KUKA KRL program: cell.src

&ACCESS RVP
&REL 20
&COMMENT 03-10-R1 AUTO EXTERNAL MAIN
DEF  CELL ( )
;********************************
; Gestamp Standards
; Line - BMW G65 (cell 03)
; Robot 03-10-R1 (BMW-03-10-R1)
; Application - AUTOMATIC EXTERNAL MAIN PROGRAM (AUTOMATIONCORE CELL)
;********************************
;FOLD Initialize System
  ;NOTE: DMY IS A REMNANT OF THE KUKA CELL TEMPLATE (cellVorgabe): WRITTEN HERE, NEVER READ
  DECL CHAR DMY[3]
  DMY[]="---"
  ;AUTOMATIONCORE START-UP (HomeCheck, PROCESS RESET), THEN PTP TO HOME (HOME.src, P1 = XHOME)
  InitializeSystem()
  HOME()
  ;ENDFOLD (Initialize System)
  LOOP
    ;FOLD Maintain System
    ;RESET CYCLE DATA AND THE PLC HANDSHAKE OUTPUTS TO THEIR REST STATE (MaintainSystem), E.G.
    ;SIGNALS $OUT[5] do005RobotInCycle OFF, $OUT[15] do015WorkComplete OFF,
    ;$OUT[4] do004ProcessFault OFF, $OUT[141] do141RedRabbitFailed OFF,
    ;$OUT[142] do142RedRabbitPassed OFF; THEN WAITS HERE WHILE STOP AT END OF CYCLE IS
    ;SELECTED (SIGNAL $IN[147] di147SEOC ON, OR SELECTED BY THE USER)
    MaintainSystem()
    ;ENDFOLD (Maintain System)
    ;FOLD Check Style
    ;READ THE STYLE NUMBER - SIGNALS $IN[33..37] gdiStyle, ECHOED ON $OUT[33..37] gdoStyleAckn
    nStyle=gdiStyle
    gdoStyleAckn=nStyle
    ;READ THE OPTION NUMBER - SIGNALS $IN[38..45] gdiOption, ECHOED ON $OUT[38..45] gdoOptionAckn
    nOption=gdiOption
    gdoOptionAckn=nOption
    ;DECODE nOption INTO bOption1..8 (GetOptions) AND WRITE THEM TO
    ;SIGNALS $OUT[38..45] do038OptionAckn1..do045OptionAckn8
    GetOptions( )
    ;SHOW THE LAST CYCLE TIME AS A STATE MESSAGE
    GetCycTime( )
    ;FOLD State Message - Waiting for Cycle Start or Style Selection.
    IF (Exists_KrlMsg(nCycleStart_Handle)==FALSE) THEN
    	nCycleStart_Handle = Set_Krlmsg (#STATE, AutomationCore_Msg[24], AutoCore_MsgPar[], AutoCore_MsgOpt_NoStop)
    ENDIF
    ;ENDFOLD (State Message - Waiting for Cycle Start or Style Selection.)
    ;ENDFOLD (Check Style)
    ;CYCLE START - SIGNAL $IN[5] di005InitiateCycle ON, WITH nStyle > 0 AND nOption > 0
    IF ((di005InitiateCycle==TRUE) AND (nStyle>0) AND (nOption>0)) THEN
	    ;FOLD Start Cycle
	    ;CLEAR AUTOMATIONCORE MESSAGES, THEN HomeCheck: THE ROBOT MUST BE AT HOME
	    ;(IF NOT: PounceToHome WHEN AT POUNCE IN EXT, OTHERWISE AN OPERATOR DIALOG)
	    AC_Erase( )
	    HomeCheck( )
	    ;ROBOT IN CYCLE - SIGNAL $OUT[5] do005RobotInCycle ON
	    do005RobotInCycle = TRUE
	    ;START THE CYCLE TIMER
	    StartCycTime( )
	    ;ENDFOLD (Start Cycle)
	    ;SELECT THE STYLE PROGRAM BY STYLE NUMBER nStyle (gdiStyle); ONLY STYLE 1 EXISTS
	    SWITCH  nStyle
		    CASE 1
             ;STYLE 1 PROGRAM
             Style_1( )
		    DEFAULT
		    ;NOTE: ANY OTHER STYLE RUNS NOTHING AND THE CYCLE ENDS AS IF COMPLETE (F06)
	    ENDSWITCH
	    ;FOLD Finish Cycle
       IF ((nStyle>0) AND (nOption>0)) THEN
		    ;END OF CYCLE (EndOfCycle)
		    ;WARNING: THE VENDOR ROUTINE EndOfCycle WAS EDITED ON THIS ROBOT: IT NO LONGER SETS
		    ;  $OUT[15] do015WorkComplete NOR WAITS FOR $IN[15] di015WorkCompleteAckn - THE PLC
		    ;  NEVER RECEIVES WORK COMPLETE FROM THIS ROBOT (F46)
		    EndOfCycle( )
		    ;STOP THE CYCLE TIMER
		    StopCycTime( )
        ENDIF
	  	;ENDFOLD (Finish Cycle)
  	ELSE
		  ;NO VALID CYCLE START - SERVICE REQUESTS FROM THE PLC (REPAIR, MASTERING REFERENCE,
		  ;BRAKE TEST, ELECTRODE CHANGE)
		  ;GO TO REPAIR - SIGNAL $IN[9] di009GoToRepair ON
		  IF (di009GoToRepair==TRUE) THEN
		  	HomeCheck( )
		  	HomeToRepair( )
;WAIT FOR RETURN FROM REPAIR - SIGNAL $IN[8] di008ReturnFromRepair ON (NO TIMEOUT, F15)
;FOLD WAIT FOR ( IN 8 'di008ReturnFromRepair' );%{PE}%R 8.3.43,%MKUKATPBASIS,%CEXT_WAIT_FOR,%VEXT_WAIT_FOR,%P 2:, 4:, 5:$IN, 6:8, 7:di008ReturnFromRepair, 9:
WAIT FOR  ( $IN[8] )
;ENDFOLD
		  		RepairToHome( )
		  ENDIF
		  ;MASTERING REFERENCE TEST - SIGNAL $IN[22] di022MstrRefRequest ON
		  IF (di022MstrRefRequest==TRUE) THEN
           HomeCheck( )
           masref_main( )
;FOLD WAIT Time=5 sec;%{PE}%R 8.3.43,%MKUKATPBASIS,%CWAIT,%VWAIT,%P 3:5
WAIT SEC 5
;ENDFOLD
		  ENDIF
          ;BRAKE TEST - SIGNAL $IN[21] di021BrakeTestRequest ON
          IF (di021BrakeTestRequest==TRUE) THEN
             HomeCheck( )
           BrakeTestReq( )
;FOLD WAIT Time=5 sec;%{PE}%R 8.3.43,%MKUKATPBASIS,%CWAIT,%VWAIT,%P 3:5
WAIT SEC 5
;ENDFOLD
        ENDIF
		  ;ELECTRODE CHANGE - SIGNAL $OUT[111] do111Gun1ElectrodeChange, $OUT[112] do112Gun2ElectrodeChange
		  ;OR $OUT[113] do113Gun3ElectrodeChange ON
		  ;NOTE: THESE ARE ROBOT OUTPUTS WRITTEN ONLY BY THE AutomationCore BACKGROUND TASK, WHICH IS
		  ;  DISABLED IN sps.sub (F12): AS IT STANDS GunElectrodeChange IS NEVER CALLED (F43)
		  IF (do111Gun1ElectrodeChange==TRUE) OR (do112Gun2ElectrodeChange==TRUE) OR (do113Gun3ElectrodeChange==TRUE) THEN
         GunElectrodeChange()
		  ENDIF
     ENDIF
  ENDLOOP
END
